Staubli VAL3: cartReceiver.pgx

public program cartReceiver()
  local bool l_bOk
  local num l_nPrefix[4]
  local num l_nHeader[12]
  local num l_nBody[52]
  local num l_nMsgType
  local num l_nPrefixLen
  local num l_nCommType
  local num l_nReplyCode
  local num l_nCartPoseType
  local num l_nPoseData[9]
  local point l_pTarget
begin
  while (true)
    l_bOk = false
    call recvData(siTcpIpCart, l_nPrefix, nCartConnFlag, l_bOk)
    if (l_bOk)
      call recvData(siTcpIpCart, l_nHeader, nCartConnFlag, l_bOk)
    endIf

    if (l_bOk)
      fromBinary(l_nHeader, 4, "-4l", l_nMsgType)

      if(l_nMsgType==nStdMsgType["CART_GET_POSE"])
        call recvData(siTcpIpCart, l_nBody, nCartConnFlag, l_bOk)
        if (l_bOk)
          nCartMsgTime = clock()
          l_pTarget = here(tTool, world)

          l_nPrefixLen = 64
          l_nCartPoseType = nStdMsgType["CART_POSE"]
          l_nCommType = 1
          l_nReplyCode = 1

          toBinary(l_nPrefixLen, 1, "-4l", l_nPrefix)
          toBinary(l_nCartPoseType, 1, "-4l", l_nHeader)
          toBinary(l_nCommType, 1, "-4l", l_nHeader[4])
          toBinary(l_nReplyCode, 1, "-4l", l_nHeader[8])

          l_nPoseData[0] = 0
          l_nPoseData[1] = l_pTarget.trsf.x * 0.001
          l_nPoseData[2] = l_pTarget.trsf.y * 0.001
          l_nPoseData[3] = l_pTarget.trsf.z * 0.001
          l_nPoseData[4] = l_pTarget.trsf.rx
          l_nPoseData[5] = l_pTarget.trsf.ry
          l_nPoseData[6] = l_pTarget.trsf.rz
          l_nPoseData[7] = 0
          l_nPoseData[8] = 0

          toBinary(l_nPoseData[0], 1, "-4l", l_nBody)
          toBinary(l_nPoseData[1], 1, "4.0l", l_nBody[4])
          toBinary(l_nPoseData[2], 1, "4.0l", l_nBody[8])
          toBinary(l_nPoseData[3], 1, "4.0l", l_nBody[12])
          toBinary(l_nPoseData[4], 1, "4.0l", l_nBody[16])
          toBinary(l_nPoseData[5], 1, "4.0l", l_nBody[20])
          toBinary(l_nPoseData[6], 1, "4.0l", l_nBody[24])
          toBinary(l_nPoseData[7], 1, "4.0l", l_nBody[28])
          toBinary(l_nPoseData[8], 1, "4.0l", l_nBody[32])

          call sendData(siTcpIpCart, l_nPrefix, nCartConnFlag)
          call sendData(siTcpIpCart, l_nHeader, nCartConnFlag)
          call sendData(siTcpIpCart, l_nBody, nCartConnFlag)
        endIf
      endIf
    endIf

    delay(0)
  endWhile
end
